TYPE ST_CoaxVisionProcessConfig :
STRUCT
    eVisionMode : E_VisionMode;
    // Simulation模式的同轴度统一结果，不参与公共通信层。
    fSimulatedCoaxiality : LREAL;
    fSimulatedDeltaX : LREAL;
    fSimulatedDeltaY : LREAL;
END_STRUCT
END_TYPE

(* stored: Version 1.1.0.1, ProductVersion 3.1.4026.20
   DUT ST_CoaxVisionProcessConfig: Id {4C8CA70C-C0FC-42A2-A613-E903E491670F} *)
